(* IEC 61131-3 sources: ae-tiax/test, 2 files *)

(* ---- CompareArray.st ---- *)
NAMESPACE Simatic.Ax.Helper
    FUNCTION CompareArray : BOOL
        VAR_INPUT
            first : ARRAY[*] OF CHAR;
            scnd : ARRAY[*] OF CHAR;
            count : INT;
        END_VAR
        VAR_TEMP
            i : DINT;
            sFirst : DINT;
            sScnd : DINT;
            eFirst : DINT;
            eScnd : DINT;
            res : BOOL;
            _count : DINT;
        END_VAR

        sFirst := LOWER_BOUND(first, 1);
        sScnd := LOWER_BOUND(scnd, 1);
        eFirst := UPPER_BOUND(first, 1);
        eScnd := UPPER_BOUND(scnd, 1);

        _count := count;

        IF ((eFirst - sFirst + 1) < count) THEN
            CompareArray := FALSE;
            RETURN;
        END_IF;
        IF ((eScnd - sScnd + 1) < count) THEN
            CompareArray := FALSE;
            RETURN;
        END_IF;

        IF _count > (eFirst - sFirst + 1) THEN
            _count := eFirst - sFirst + 1;
        END_IF;

        FOR i := 0 TO _count - 1 DO
            res := first[i + sFirst] = scnd[i + sScnd];
            IF (res = FALSE) THEN
                CompareArray := FALSE;
                RETURN;
            END_IF;
        END_FOR;
        CompareArray := TRUE;
    END_FUNCTION
END_NAMESPACE

(* ---- test.st ---- *)
USING Simatic.Ax.Tiax;
USING AxUnit;
USING Simatic.Ax.Conversion;

NAMESPACE MyTest

    {TestFixture}
    CLASS TestJsonStructure
        VAR
            o : JsonStructure;
            len : DINT;
            expString : STRING;
            cmpBuff : ARRAY[0..399] OF CHAR;
            isEqual : BOOL;
        END_VAR
        {Test}
        METHOD PUBLIC Excecute_of_the_wrapper_returns_the_Correct_JSON_String
            expString := '{"DeviceName": "Device1", "Parameter": {"IP": "192.168.0.1", "Timeout": 300, "AutoConnect": true}}';
            len := Strings.ToArray.OfCharCount(str := expString, arr := cmpBuff);

            o.DeviceName := 'Device1';
            o.IP := '192.168.0.1';
            o.Timeout := 300;
            o.AutoConnect := TRUE;
            o(Execute := TRUE);
            isEqual := Simatic.Ax.Helper.CompareArray(first := o.Result, scnd := cmpBuff, count := TO_INT(len));
            Assert.Equal(actual := isEqual, expected := TRUE);
        END_METHOD
    END_CLASS

END_NAMESPACE
